# EPICS autosave request: stdApp/Db/saveData_settings.req
$(P)saveData_fileSystem
$(P)saveData_subDir
$(P)saveData_scanNumber
